// Mitsubishi GX Works2 project: Dimaculangan, Raven_PGC   PLC: FX1N/FX1NC

PROGRAM MAIN
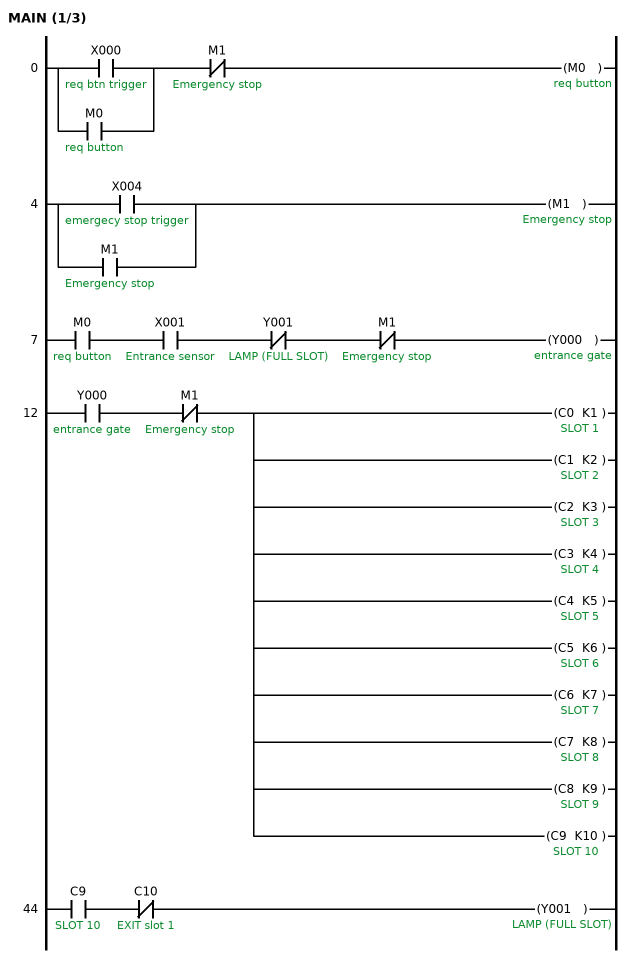
0     LD      X000  ; req btn trigger
      OR      M0  ; req button
      ANI     M1  ; Emergency stop
      OUT     M0  ; req button
4     LD      X004  ; emergecy stop trigger
      OR      M1  ; Emergency stop
      OUT     M1  ; Emergency stop
7     LD      M0  ; req button
      AND     X001  ; Entrance sensor
      ANI     Y001  ; LAMP (FULL SLOT)
      ANI     M1  ; Emergency stop
      OUT     Y000  ; entrance gate
12    LD      Y000  ; entrance gate
      ANI     M1  ; Emergency stop
      OUT     C0 K1  ; SLOT 1
      OUT     C1 K2  ; SLOT 2
      OUT     C2 K3  ; SLOT 3
      OUT     C3 K4  ; SLOT 4
      OUT     C4 K5  ; SLOT 5
      OUT     C5 K6  ; SLOT 6
      OUT     C6 K7  ; SLOT 7
      OUT     C7 K8  ; SLOT 8
      OUT     C8 K9  ; SLOT 9
      OUT     C9 K10  ; SLOT 10
44    LD      C9  ; SLOT 10
      ANI     C10  ; EXIT slot 1
      OUT     Y001  ; LAMP (FULL SLOT)
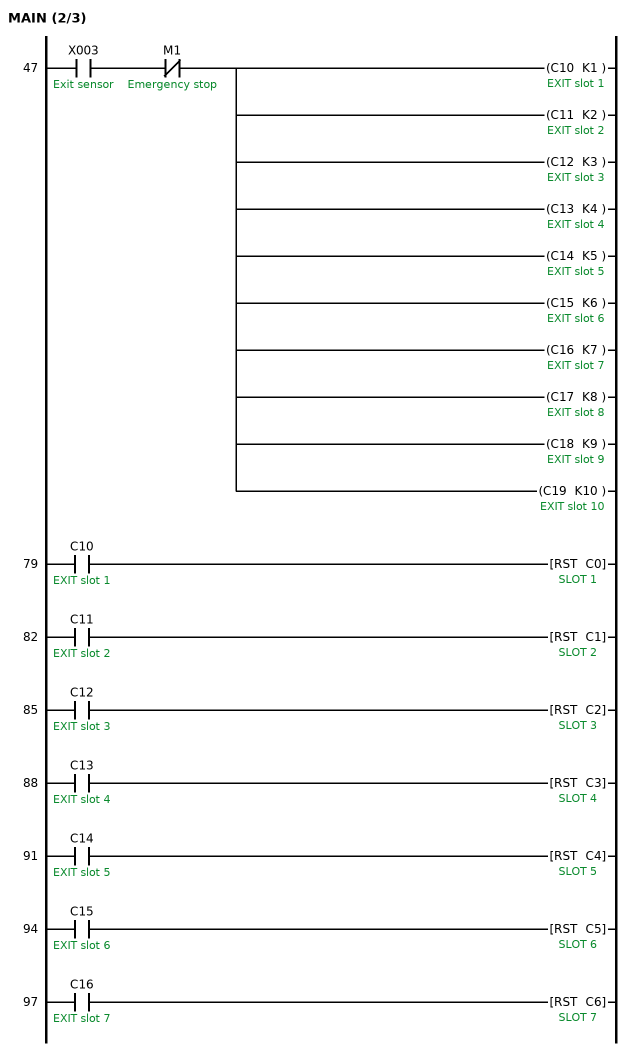
47    LD      X003  ; Exit sensor
      ANI     M1  ; Emergency stop
      OUT     C10 K1  ; EXIT slot 1
      OUT     C11 K2  ; EXIT slot 2
      OUT     C12 K3  ; EXIT slot 3
      OUT     C13 K4  ; EXIT slot 4
      OUT     C14 K5  ; EXIT slot 5
      OUT     C15 K6  ; EXIT slot 6
      OUT     C16 K7  ; EXIT slot 7
      OUT     C17 K8  ; EXIT slot 8
      OUT     C18 K9  ; EXIT slot 9
      OUT     C19 K10  ; EXIT slot 10
79    LD      C10  ; EXIT slot 1
      RST     C0  ; SLOT 1
82    LD      C11  ; EXIT slot 2
      RST     C1  ; SLOT 2
85    LD      C12  ; EXIT slot 3
      RST     C2  ; SLOT 3
88    LD      C13  ; EXIT slot 4
      RST     C3  ; SLOT 4
91    LD      C14  ; EXIT slot 5
      RST     C4  ; SLOT 5
94    LD      C15  ; EXIT slot 6
      RST     C5  ; SLOT 6
97    LD      C16  ; EXIT slot 7
      RST     C6  ; SLOT 7
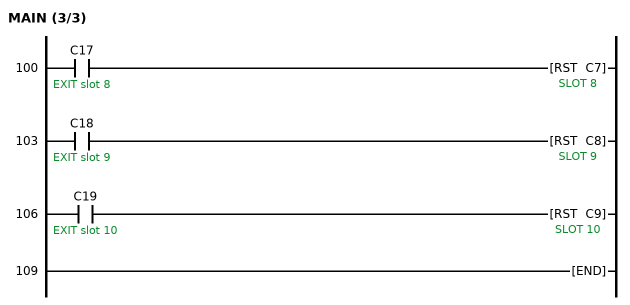
100   LD      C17  ; EXIT slot 8
      RST     C7  ; SLOT 8
103   LD      C18  ; EXIT slot 9
      RST     C8  ; SLOT 9
106   LD      C19  ; EXIT slot 10
      RST     C9  ; SLOT 10
109   END
END_PROGRAM

// device comments not shown above
X002  ; entry of car
